// TIA Portal V17 export
// export: Created 2026-08-11T13:54:29.0707996Z, ExportSetting WithDefaults, DisplayName Totally Integrated Automation Portal, DisplayVersion V17, DisplayName TIA Portal Openness, DisplayVersion V17, DisplayName TIA Portal Version Control Interface, DisplayVersion V17, DisplayName STEP 7 Professional, DisplayVersion V17, DisplayName STEP 7 Safety, DisplayVersion V17, DisplayName WinCC Professional, DisplayVersion V17
Screen "总画面"  1280x800, Number=1, Template=模板_2
  ScreenLayer 
    GraphicView "背景图片" at 0,100 size 1278x700  Picture=QQ截图20160302143524
    Button "按钮_3" at 761,584 size 48x29  Mode=Text, TextOn="Text"
    Button "按钮_2" at 216,380 size 215x92  Mode=Text, TextOff="成品库", TextOn="Text"
      on Release: ActivateScreen(Screen name := 成品库, Object number := 0)
    Button "按钮_6" at 832,379 size 215x92  Mode=Text, TextOff="报警查询", TextOn="Text"
      on Release: ActivateScreen(Screen name := 故障查询画面, Object number := 0)
    Button "按钮_7" at 526,377 size 215x92  Mode=Text, TextOff="权限管理", TextOn="Text"
      on Release: ActivateScreen(Screen name := 权限管理画面, Object number := 0)
